// TwinCAT 3 PLC project Plc
// ProgramVersion: 3.1.4026.19
// libraries:
//   Tc2_Standard, * (Beckhoff Automation GmbH)
//   Tc2_System, * (Beckhoff Automation GmbH)
//   TcUnit, * (www.tcunit.org)
// project tree:
//   / CCTask1.TcTTO, CCTask2.TcTTO, PlcTask.TcTTO
//   Program/ MAIN.TcPOU
//   Src/Base/ FB_VarByteBufferBase.TcPOU, I_VarByteBufferBase.TcIO
//   Src/SimpleDynBuffer/ FB_SimpleRingBuffer.TcPOU, I_SimpleRingBuffer.TcIO
//   Src/ThreadSafe/ FB_SpscBuffer.TcPOU, I_SpscBuffer.TcIO
//   Src/VarByteBuffer/ FB_VarByteBuffer.TcPOU, I_VarByteBuffer.TcIO
//   Src/VarStringBuffer/ FB_VarStringBuffer.TcPOU, I_VarStringBuffer.TcIO
//   _test/SimpleRingBuffer/DUT/ ST_TestStruct.TcDUT
//   _test/SimpleRingBuffer/ FB_TestSimpleDynBuffer.TcPOU
//   _test/ThreadSafe/ ProgramTask1.TcPOU, ProgramTask2.TcPOU
//   _test/VarStringBuffer/ FB_TestVarStringBuffer.TcPOU
// real-time tasks:
//   TASK PlcTask: cycle T#30ms, priority 20, ADS port 350
//   TASK CCTask1: cycle T#2ms, priority 1, ADS port 351
//   TASK CCTask2: cycle T#3ms, priority 2, ADS port 352

CONFIGURATION Plc
    RESOURCE PLC ON TwinCAT3
        TASK CCTask1(INTERVAL := T#2ms, PRIORITY := 1);
        TASK CCTask2(INTERVAL := T#3ms, PRIORITY := 2);
        TASK PlcTask(INTERVAL := T#30ms, PRIORITY := 20);
        PROGRAM ProgramTask1 WITH CCTask1 : ProgramTask1;
        PROGRAM ProgramTask2 WITH CCTask2 : ProgramTask2;
        PROGRAM MAIN WITH PlcTask : MAIN;
    END_RESOURCE
END_CONFIGURATION

// ---- _test/SimpleRingBuffer/DUT/ST_TestStruct.TcDUT
TYPE ST_TestStruct :
STRUCT
	nIndex: UDINT;
	aData : ARRAY[1..1020] OF BYTE;
END_STRUCT
END_TYPE

// ---- Src/Base/I_VarByteBufferBase.TcIO
INTERFACE I_VarByteBufferBase

PROPERTY Buffer : PVOID
GET
END_GET
END_PROPERTY

PROPERTY Capacity : UDINT
GET
END_GET
END_PROPERTY

METHOD Clear : BOOL
END_METHOD

PROPERTY FreeBytes : UDINT
GET
END_GET
END_PROPERTY

METHOD Initialize : BOOL
VAR_INPUT
	nBufferSize 		: UDINT; // Size in byte
END_VAR
END_METHOD

METHOD Reset
END_METHOD

PROPERTY Size : UDINT
GET
END_GET
END_PROPERTY

END_INTERFACE

// ---- Src/SimpleDynBuffer/I_SimpleRingBuffer.TcIO
INTERFACE I_SimpleRingBuffer

PROPERTY Capacity : UDINT
GET
END_GET
END_PROPERTY

PROPERTY Empty : bool
GET
END_GET
END_PROPERTY

PROPERTY Full : bool
GET
END_GET
END_PROPERTY

METHOD Get : BOOL
VAR_INPUT
	pDestination 	: pvoid;
	cbSize 			: UDINT;
END_VAR
END_METHOD

METHOD Initialize : BOOL
VAR_INPUT
	nElementSize 		: UDINT;
	nElementCapacity 	: UDINT;
END_VAR
END_METHOD

METHOD Push : BOOL
VAR_INPUT
	pData : pvoid;
	cbSize : UDINT;
END_VAR
END_METHOD

METHOD Reset
END_METHOD

PROPERTY Size : UDINT
GET
END_GET
END_PROPERTY

END_INTERFACE

// ---- Src/ThreadSafe/I_SpscBuffer.TcIO
INTERFACE I_SpscBuffer

PROPERTY Capacity : UDINT
GET
END_GET
END_PROPERTY

METHOD Clear
VAR_INPUT
END_VAR
END_METHOD

PROPERTY Empty : bool
GET
END_GET
END_PROPERTY

PROPERTY Full : bool
GET
END_GET
END_PROPERTY

METHOD Get : BOOL
VAR_INPUT
	pDestination 	: pvoid;
	cbSize 			: UDINT;
END_VAR
END_METHOD

METHOD Initialize : BOOL
VAR_INPUT
	nElementSize 		: UDINT;
	nElementCapacity 	: UDINT;
END_VAR
END_METHOD

METHOD Push : BOOL
VAR_INPUT
	pData : pvoid;
	cbSize : UDINT;
END_VAR
END_METHOD

METHOD Reset
END_METHOD

PROPERTY Size : UDINT
GET
END_GET
END_PROPERTY

END_INTERFACE

// ---- Src/VarByteBuffer/I_VarByteBuffer.TcIO
INTERFACE I_VarByteBuffer EXTENDS I_VarByteBufferBase

METHOD Push : BOOL
VAR_INPUT
	pData : pvoid;
	cbSize : UDINT;
END_VAR
END_METHOD

END_INTERFACE

// ---- Src/VarStringBuffer/I_VarStringBuffer.TcIO
INTERFACE I_VarStringBuffer EXTENDS I_VarByteBufferBase

METHOD Push : BOOL
VAR_INPUT
	sInputString	: REFERENCE TO T_MaxString;
END_VAR
END_METHOD

END_INTERFACE

// ---- _test/ThreadSafe/ProgramTask1.TcPOU
PROGRAM ProgramTask1
VAR
	fbSpscBuff 	: FB_SpscBuffer;
	ipSpscBuff 	: I_SpscBuffer 		:= fbSpscBuff;
	nCounter 	: UDINT;
	bInit 		: BOOL;
END_VAR

nCounter := nCounter + 1;
IF NOT(binit) THEN
	bInit := TRUE;
	ipSpscBuff.Initialize(SIZEOF(UDINT),100);
END_IF

ipSpscBuff.Push(ADR(nCounter),SIZEOF(nCounter));
ipSpscBuff.Reset();

END_PROGRAM

// ---- Src/ThreadSafe/FB_SpscBuffer.TcPOU
FUNCTION_BLOCK FB_SpscBuffer IMPLEMENTS I_SpscBuffer
VAR
	_pBuffer 		: POINTER TO BYTE;
	_nTail 			: UDINT;
	_nHead 			: UDINT;
	_nCapacity 		: UDINT;
	_bFull 			: BOOL;
	_nSize 			: UDINT;
	
	_fbCriticalSection : FB_IecCriticalSection;
	_nElementSize 	: UDINT;
	_nLockFailures	: UDINT;
	_nError 		: UDINT;
END_VAR
VAR CONSTANT
	cMaxElementSize : UDINT := 4096;
END_VAR

PROPERTY Capacity : UDINT
GET
Capacity := this^._nCapacity;
END_GET
END_PROPERTY

METHOD Clear
VAR_INPUT
END_VAR
IF THIS^._fbCriticalSection.Enter() THEN
	THIS^._nTail 			:= 0;
	THIS^._nHead 			:= 0;
	THIS^._nCapacity 		:= 0;
	THIS^._bFull 			:= 0;
	THIS^._nSize 			:= 0;
	THIS^._nElementSize 	:= 0;
	THIS^._nError 			:= 0;
	THIS^._fbCriticalSection.Leave();
ELSE
	THIS^._nLockFailures := THIS^._nLockFailures :=  + 1;
	RETURN;
END_IF
END_METHOD

PROPERTY Empty : bool
GET
Empty := not(this^._bFull) and (this^._nHead = this^._nTail);
END_GET
END_PROPERTY

//FB_Exit must be implemented explicitly. If there is an implementation, then the
//method is called before the controller removes the code of the function block instance
//(implicit call). The return value is not evaluated.
METHOD FB_Exit: BOOL
VAR_INPUT
    bInCopyCode: BOOL;  // TRUE: the exit method is called in order to leave the instance which will be copied afterwards (online change).  
END_VAR
this^.Reset();
END_METHOD

PROPERTY Full : bool
GET
Full := this^._bFull;
END_GET
END_PROPERTY

METHOD Get : BOOL
VAR_INPUT
	pDestination 	: pvoid;
	cbSize 			: UDINT;
END_VAR
VAR
	nByteOffset : UDINT;
	res 		: UDINT;
END_VAR
IF THIS^._fbCriticalSection.Enter() THEN
	IF (THIS^._pBuffer = 0) OR (THIS^._nCapacity = 0) THEN  RETURN; END_IF; 	// Check initialization
	IF pDestination = 0 THEN  RETURN; END_IF;								// Check input
	IF cbSize <> THIS^._nElementSize THEN  RETURN; END_IF;					// Check input
	IF THIS^.Empty THEN RETURN; END_IF;										// Check internal state
	
	nByteOffset := THIS^._nTail*THIS^._nElementSize;
	res := memcpy(pDestination, THIS^._pBuffer + nByteOffset, THIS^._nElementSize);
	
	IF res <> THIS^._nElementSize THEN
		THIS^._nError := THIS^._nError + 1;
	END_IF
	
	THIS^._bFull := FALSE;
	IF THIS^._nSize > 0 THEN
		THIS^._nSize := THIS^._nSize - 1;	
	END_IF
	THIS^._nTail := (THIS^._nTail + 1) MOD THIS^._nCapacity;
	
	THIS^._fbCriticalSection.Leave();
	Get := TRUE;

ELSE
	THIS^._nLockFailures := THIS^._nLockFailures :=  + 1;
	RETURN;
END_IF
END_METHOD

METHOD Initialize : BOOL
VAR_INPUT
	nElementSize 		: UDINT;
	nElementCapacity 	: UDINT;
END_VAR
VAR
	nSize 				: UDINT;
END_VAR
IF nElementSize = 0 OR nElementCapacity = 0 THEN RETURN; END_IF;
IF nElementSize > THIS^.cMaxElementSize THEN RETURN; END_IF;
IF (nElementCapacity > (TO_UDINT(16#FFFFFFFF) / nElementSize)) THEN RETURN; END_IF;

THIS^.Reset();

nSize := nElementSize * nElementCapacity;
THIS^._pBuffer := __NEW(BYTE, nSize);

IF THIS^._pBuffer = 0 THEN RETURN; END_IF;
THIS^._nElementSize := nElementSize;
THIS^._nCapacity := nElementCapacity;
Initialize := TRUE;
END_METHOD

METHOD Push : BOOL
VAR_INPUT
	pData : pvoid;
	cbSize : UDINT;
END_VAR
VAR
	nByteOffset : UDINT;
	res			: UDINT;
END_VAR
IF THIS^._fbCriticalSection.Enter() THEN
	
	IF (THIS^._pBuffer = 0) OR (THIS^._nCapacity = 0) THEN RETURN; END_IF;		// Check initialization
	IF THIS^._bFull THEN RETURN; END_IF;
	IF cbSize <> THIS^._nElementSize THEN RETURN; END_IF;						// Check input
	IF pData = 0 THEN RETURN; END_IF											// Check input
	
	nByteOffset := THIS^._nHead*THIS^._nElementSize;
	res := memcpy(THIS^._pBuffer + nByteOffset,pData,THIS^._nElementSize);
	IF res <> THIS^._nElementSize THEN
		THIS^._nError := THIS^._nError + 1; 
	END_IF	

	THIS^._nSize := THIS^._nSize + 1;

	
	THIS^._nHead := (THIS^._nHead + 1) MOD THIS^._nCapacity;
	THIS^._bFull := THIS^._nHead = THIS^._nTail;
	
	Push := TRUE;
	THIS^._fbCriticalSection.Leave();
	

ELSE
	THIS^._nLockFailures := THIS^._nLockFailures :=  + 1;
	RETURN;
END_IF
END_METHOD

METHOD Reset
IF THIS^._fbCriticalSection.Enter() THEN
	IF THIS^._pBuffer <> 0 THEN
		__DELETE(THIS^._pBuffer);
		THIS^._pBuffer := 0;
	END_IF
	
	THIS^._nTail 			:= 0;
	THIS^._nHead 			:= 0;
	THIS^._nCapacity 		:= 0;
	THIS^._bFull 			:= 0;
	THIS^._nSize 			:= 0;
	THIS^._nElementSize 	:= 0;
	THIS^._nError 			:= 0;
	THIS^._fbCriticalSection.Leave();
ELSE
	THIS^._nLockFailures := THIS^._nLockFailures :=  + 1;
	RETURN;
END_IF
END_METHOD

PROPERTY Size : UDINT
GET
Size := (this^._nHead-this^._nTail + this^.Capacity) mod this^.Capacity;
END_GET
END_PROPERTY

END_FUNCTION_BLOCK

// ---- _test/ThreadSafe/ProgramTask2.TcPOU
PROGRAM ProgramTask2
VAR
	nRead : udint;
END_VAR

ProgramTask1.ipSpscBuff.Get(ADR(nRead),SIZEOF(nRead));

END_PROGRAM

// ---- Program/MAIN.TcPOU
PROGRAM MAIN
VAR
	nCounter 				: INT;
	fbTestSimpleDynBuffer 	: FB_TestSimpleDynBuffer;
	fbTestVarByteBuffer		: FB_TestVarStringBuffer;
END_VAR

nCounter := nCounter + 1;

TcUnit.RUN();

END_PROGRAM

// ---- _test/SimpleRingBuffer/FB_TestSimpleDynBuffer.TcPOU
FUNCTION_BLOCK FB_TestSimpleDynBuffer EXTENDS TcUnit.FB_TestSuite
VAR

	// FillTenElements
	fbBufferTest1 : FB_SimpleRingBuffer;
	ipBufferTest1 : I_SimpleRingBuffer := fbBufferTest1;

	//OverflowOneElement
	fbBufferTest2 : FB_SimpleRingBuffer;
	ipBufferTest2 : I_SimpleRingBuffer := fbBufferTest2;

	//ResetAndUse
	fbBufferTest3 : FB_SimpleRingBuffer;
	ipBufferTest3 : I_SimpleRingBuffer := fbBufferTest2;

	//CheckMemoryLeaks
	fbBufferTest4 	: FB_SimpleRingBuffer;
	ipBufferTest4 	: I_SimpleRingBuffer := fbBufferTest4;
	nState4 		: UDINT;
	nFillPerCycle 	: UDINT := 64;
	nKbToFill 		: UDINT := 10*1024;
	nFillCyclesToDo : UDINT := nKbToFill/nFillPerCycle; // 10 mb 
	nFillCycle 		: UDINT;
	nErrors4 		: UDINT;

	//CheckInvalidInput
	fbBufferTest5 : FB_SimpleRingBuffer;
	ipBufferTest5 : I_SimpleRingBuffer := fbBufferTest2;

END_VAR

FillTenElements();
OverflowOneElement();
ResetAndUse();
// CheckMemoryLeaks();
CheckInvalidInput();

METHOD CheckInvalidInput : REFERENCE TO FB_Test
VAR
	i 		: UDINT;
	nGet : UDINT;

END_VAR
TEST('CheckInvalidInput');


IF ipBufferTest5.Initialize(	nElementSize := 0,
								nElementCapacity := 1) THEN
	AssertTrue(FALSE, 'Failed init 0 element size');		
END_IF;

IF ipBufferTest5.Initialize(	nElementSize := 4,
								nElementCapacity := 0) THEN
	AssertTrue(FALSE, 'Failed init 0 capacity');		
END_IF;

IF NOT ipBufferTest5.Initialize(	nElementSize := 4,
									nElementCapacity := 1) THEN
	AssertTrue(FALSE, 'Failed init');		
END_IF;

IF ipBufferTest5.Push(ADR(i),0) THEN
	AssertTrue(FALSE, 'Failed push size 0');		
END_IF

IF ipBufferTest5.Push(0,4) THEN
	AssertTrue(FALSE, 'Failed push adr 0');		
END_IF

IF NOT ipBufferTest5.Push(ADR(i),4) THEN
	AssertTrue(FALSE, 'Failed push legit data');		
END_IF

IF ipBufferTest5.Get(ADR(i),0) THEN
	AssertTrue(FALSE, 'Failed get size 0');		
END_IF

IF ipBufferTest5.Get(0,4) THEN
	AssertTrue(FALSE, 'Failed get adr 0');		
END_IF

TEST_FINISHED();
END_METHOD

METHOD CheckMemoryLeaks : REFERENCE TO FB_Test
VAR
	i,j 				: UDINT;
	nElementsSize 		: UDINT;
	nOverflow			: UDINT 	:= 2;
	stDataToInsert		: ST_TestStruct; // 1024 bytes
	nElementsToPush		:UDINT;
	nReadSize 			: UDINT;
	bIsFull 			: BOOL;
	bIsEmpty 			: BOOL;
	nReadCapacity		: UDINT;
	
	nGetValue : ST_TestStruct;
	
	nExpectedValue : UDINT;
END_VAR
TEST('CheckMemoryLeaks');

CASE nState4 OF 
	0:

		nElementsSize := SIZEOF(ST_TestStruct);
		IF NOT fbBufferTest4.Initialize(	nElementSize := nElementsSize,
											nElementCapacity := 1024*10) THEN
 			nErrors4 := nErrors4 +1;
		END_IF;
		nState4 := 1;			
		

	1:
		IF nFillCycle = nFillCyclesToDo THEN
			nElementsToPush := nFillPerCycle + nOverflow;
		ELSE
			nElementsToPush := nFillPerCycle;
		END_IF
		FOR i := 1 TO nElementsToPush DO
			stDataToInsert.nIndex := i;
			IF NOT fbBufferTest4.Push(ADR(stDataToInsert), SIZEOF(stDataToInsert)) THEN
				nErrors4 := nErrors4 +1;
			END_IF
		END_FOR
		nFillCycle := nFillCycle + 1;
		IF nFillCycle >= nFillCyclesToDo THEN
			nFillCycle := 1;
			nState4 := 10;
		END_IF
	10:
		// Free cylce
		FOR i := 1 TO nFillPerCycle DO
			IF NOT fbBufferTest4.Get(ADR(nGetValue), SIZEOF(nGetValue)) THEN
				nErrors4 := nErrors4 +1;
			END_IF
		END_FOR

		nFillCycle := nFillCycle + 1;
		IF nFillCycle >= nFillCyclesToDo THEN
			fbBufferTest4.Reset();
			nFillCycle := 0;
			nState4 := 20;
		END_IF
	20: 
		
		bIsFull 	:= fbBufferTest4.Full;
		nReadSize 	:= fbBufferTest4.Size;
		nExpectedValue := 0;
		AssertFalse(bIsFull, 'Inconsistent Full flag');		
		AssertEquals(Expected 	:= nExpectedValue,
					 Actual 	:= nReadSize,
					 Message 	:= 'Error computing Size');		
		AssertEquals(Expected 	:= nExpectedValue,
					 Actual 	:= nErrors4,
					 Message 	:= 'Error computing Size');		
		TEST_FINISHED(); 
END_CASE
END_METHOD

METHOD FillTenElements : BOOL
VAR
	i 					: UDINT;
	nCapacity 			: UDINT 	:= 10;
	nElementsSize 		: UDINT;
	
	nReadSize 			: UDINT;
	bIsFull 			: BOOL;
	bIsEmpty 			: BOOL;
	nReadCapacity		: UDINT;
END_VAR
TEST('PushTenElements');

nElementsSize := SIZEOF(UDINT);
IF NOT ipBufferTest1.Initialize(	nElementSize := nElementsSize,
									nElementCapacity := nCapacity) THEN
	AssertTrue(FALSE, 'PushTenElements failed to initialize.');		
END_IF;

bIsEmpty := ipBufferTest1.Empty;
nReadCapacity := ipBufferTest1.Capacity;
AssertTrue(bIsEmpty, 'PushTenElements failed to initialize.');
AssertEquals(Expected 	:= nCapacity,
             Actual 	:= nReadCapacity,
             Message 	:= 'Error computing capacity');				
			 
FOR i := 1 TO nCapacity DO
	IF NOT ipBufferTest1.Push(ADR(i), SIZEOF(i)) THEN
		AssertTrue(FALSE, 'Failed to push');
	END_IF
END_FOR

bIsFull 	:= ipBufferTest1.Full;
nReadSize 	:= ipBufferTest1.Size;

AssertTrue(bIsFull, 'Inconsistent Full flag');		
AssertEquals(Expected 	:= nCapacity,
             Actual 	:= nReadSize,
             Message 	:= 'Error computing Size');		
 
TEST_FINISHED();
END_METHOD

METHOD OverflowOneElement : REFERENCE TO FB_Test
VAR
	i 					: UDINT;
	nCapacity 			: UDINT 	:= 10;
	nElementsSize 		: UDINT;
	nOverflow			: UDINT 	:= 1;
	
	nReadSize 			: UDINT;
	bIsFull 			: BOOL;
	bIsEmpty 			: BOOL;
	nReadCapacity		: UDINT;
	
	nGetValue : UDINT;
	
	nExpectedValue : UDINT;
END_VAR
TEST('OverflowOneElement');

nElementsSize := SIZEOF(UDINT);
IF NOT ipBufferTest2.Initialize(	nElementSize := nElementsSize,
									nElementCapacity := nCapacity) THEN
	AssertTrue(FALSE, 'PushTenElements failed to initialize.');		
END_IF;

bIsEmpty := ipBufferTest2.Empty;
nReadCapacity := ipBufferTest2.Capacity;
AssertTrue(bIsEmpty, 'PushTenElements failed to initialize.');
AssertEquals(Expected 	:= nCapacity,
             Actual 	:= nReadCapacity,
             Message 	:= 'Error computing capacity');				
			 
FOR i := 1 TO nCapacity + nOverflow DO
	IF NOT ipBufferTest2.Push(ADR(i), SIZEOF(i)) THEN
		AssertTrue(FALSE, 'Failed to push');
	END_IF
END_FOR
FOR i := 1 TO nCapacity DO
	IF NOT ipBufferTest2.Get(ADR(nGetValue), SIZEOF(nGetValue)) THEN
		AssertTrue(FALSE, 'Failed to get');
	ELSE
		nExpectedValue := i + nOverflow;
		AssertEquals(Expected 	:= nExpectedValue,
					 Actual 	:= nGetValue,
					 Message 	:= 'Error on Get');
	END_IF
END_FOR

bIsFull 	:= ipBufferTest2.Full;
nReadSize 	:= ipBufferTest2.Size;

nExpectedValue := 0;
AssertFalse(bIsFull, 'Inconsistent Full flag');		
AssertEquals(Expected 	:= nExpectedValue,
             Actual 	:= nReadSize,
             Message 	:= 'Error computing Size');		
 
TEST_FINISHED();
END_METHOD

METHOD ResetAndUse : REFERENCE TO FB_Test
VAR
	i,j 				: UDINT;
	nCapacity 			: UDINT 	:= 10;
	nElementsSize 		: UDINT;
	nOverflow			: UDINT 	:= 1;
	
	nReadSize 			: UDINT;
	bIsFull 			: BOOL;
	bIsEmpty 			: BOOL;
	nReadCapacity		: UDINT;
	
	nGetValue : UDINT;
	
	nExpectedValue : UDINT;
END_VAR
TEST('ResetAndUse');

FOR j := 1 TO 100 DO

	nElementsSize := SIZEOF(UDINT);
	IF NOT ipBufferTest3.Initialize(	nElementSize := nElementsSize,
										nElementCapacity := nCapacity) THEN
		AssertTrue(FALSE, 'Failed to initialize.');		
	END_IF;
	
	bIsEmpty := ipBufferTest3.Empty;
	nReadCapacity := ipBufferTest3.Capacity;
	AssertTrue(bIsEmpty, 'Failed to initialize.');
	AssertEquals(Expected 	:= nCapacity,
				 Actual 	:= nReadCapacity,
				 Message 	:= 'Error computing capacity');				
				 
	FOR i := 1 TO nCapacity + nOverflow DO
		IF NOT ipBufferTest3.Push(ADR(i), SIZEOF(i)) THEN
			AssertTrue(FALSE, 'Failed to push');
		END_IF
	END_FOR
	FOR i := 1 TO nCapacity DO
		IF NOT ipBufferTest3.Get(ADR(nGetValue), SIZEOF(nGetValue)) THEN
			AssertTrue(FALSE, 'Failed to get');
		ELSE
			nExpectedValue := i + nOverflow;
			AssertEquals(Expected 	:= nExpectedValue,
						 Actual 	:= nGetValue,
						 Message 	:= 'Error on Get');
		END_IF
	END_FOR
	
	bIsFull 	:= ipBufferTest3.Full;
	nReadSize 	:= ipBufferTest3.Size;
	
	nExpectedValue := 0;
	AssertFalse(bIsFull, 'Inconsistent Full flag');		
	AssertEquals(Expected 	:= nExpectedValue,
				 Actual 	:= nReadSize,
				 Message 	:= 'Error computing Size');		
	ipBufferTest3.Reset();
END_FOR
TEST_FINISHED();
END_METHOD

END_FUNCTION_BLOCK

// ---- Src/SimpleDynBuffer/FB_SimpleRingBuffer.TcPOU
FUNCTION_BLOCK FB_SimpleRingBuffer implements I_SimpleRingBuffer
VAR
	_pBuffer 		: POINTER TO BYTE;
	_nTail 			: UDINT;
	_nHead 			: UDINT;
	_nCapacity 		: UDINT;
	_bFull 			: BOOL;
	_nSize 			: UDINT;
	
	_nElementSize 	: UDINT;
	_nError 		: UDINT;
END_VAR
VAR CONSTANT
	cMaxElementSize : UDINT := 4096;
END_VAR

PROPERTY Capacity : UDINT
GET
Capacity := this^._nCapacity;
END_GET
END_PROPERTY

PROPERTY Empty : bool
GET
Empty := not(this^._bFull) and (this^._nHead = this^._nTail);
END_GET
END_PROPERTY

//FB_Exit must be implemented explicitly. If there is an implementation, then the
//method is called before the controller removes the code of the function block instance
//(implicit call). The return value is not evaluated.
METHOD FB_Exit: BOOL
VAR_INPUT
    bInCopyCode: BOOL;  // TRUE: the exit method is called in order to leave the instance which will be copied afterwards (online change).  
END_VAR
this^.Reset();
END_METHOD

PROPERTY Full : bool
GET
Full := this^._bFull;
END_GET
END_PROPERTY

METHOD Get : BOOL
VAR_INPUT
	pDestination 	: pvoid;
	cbSize 			: UDINT;
END_VAR
VAR
	nByteOffset : UDINT;
	res 		: UDINT;
END_VAR
IF (THIS^._pBuffer = 0) OR (THIS^._nCapacity = 0) THEN RETURN; END_IF; 	// Check initialization
IF pDestination = 0 THEN RETURN; END_IF;								// Check input
IF cbSize <> THIS^._nElementSize THEN RETURN; END_IF;					// Check input
IF THIS^.Empty THEN RETURN; END_IF;										// Check internal state

nByteOffset := THIS^._nTail*THIS^._nElementSize;
res := memcpy(pDestination, THIS^._pBuffer + nByteOffset, THIS^._nElementSize);

IF res <> THIS^._nElementSize THEN
	THIS^._nError := THIS^._nError + 1;
	RETURN;
END_IF

THIS^._bFull := FALSE;
IF THIS^._nSize > 0 THEN
	THIS^._nSize := THIS^._nSize - 1;	
END_IF
THIS^._nTail := (THIS^._nTail + 1) MOD THIS^._nCapacity;

Get := TRUE;
END_METHOD

METHOD Initialize : BOOL
VAR_INPUT
	nElementSize 		: UDINT;
	nElementCapacity 	: UDINT;
END_VAR
VAR
	nSize 				: UDINT;
END_VAR
IF nElementSize = 0 OR nElementCapacity = 0 THEN RETURN; END_IF;
IF nElementSize > THIS^.cMaxElementSize THEN RETURN; END_IF;
IF (nElementCapacity > (TO_UDINT(16#FFFFFFFF) / nElementSize)) THEN RETURN; END_IF;

THIS^.Reset();

nSize := nElementSize * nElementCapacity;
THIS^._pBuffer := __NEW(BYTE, nSize);

IF THIS^._pBuffer = 0 THEN RETURN; END_IF;
THIS^._nElementSize := nElementSize;
THIS^._nCapacity := nElementCapacity;
Initialize := TRUE;
END_METHOD

METHOD Push : BOOL
VAR_INPUT
	pData : pvoid;
	cbSize : UDINT;
END_VAR
VAR
	nByteOffset : UDINT;
	res			: UDINT;
END_VAR
IF (THIS^._pBuffer = 0) OR (THIS^._nCapacity = 0) THEN RETURN; END_IF;		// Check initialization
IF cbSize <> THIS^._nElementSize THEN RETURN; END_IF;						// Check input
IF pData = 0 THEN RETURN; END_IF											// Check input

nByteOffset := THIS^._nHead*THIS^._nElementSize;
res := memcpy(THIS^._pBuffer + nByteOffset,pData,THIS^._nElementSize);
IF res <> THIS^._nElementSize THEN
	THIS^._nError := THIS^._nError + 1; 
	RETURN;
END_IF

IF THIS^._bFull THEN
	THIS^._nTail := (THIS^._nTail + 1) MOD THIS^._nCapacity;
ELSE
	THIS^._nSize := THIS^._nSize + 1;
END_IF

THIS^._nHead := (THIS^._nHead + 1) MOD THIS^._nCapacity;
THIS^._bFull := THIS^._nHead = THIS^._nTail;

Push := TRUE;
END_METHOD

METHOD Reset
IF THIS^._pBuffer <> 0 THEN
	__DELETE(THIS^._pBuffer);
	THIS^._pBuffer := 0;
END_IF

THIS^._nTail 			:= 0;
THIS^._nHead 			:= 0;
THIS^._nCapacity 		:= 0;
THIS^._bFull 			:= 0;
THIS^._nSize 			:= 0;
THIS^._nElementSize 	:= 0;
THIS^._nError 			:= 0;
END_METHOD

PROPERTY Size : UDINT
GET
Size := this^._nSize;
END_GET
END_PROPERTY

END_FUNCTION_BLOCK

// ---- _test/VarStringBuffer/FB_TestVarStringBuffer.TcPOU
FUNCTION_BLOCK FB_TestVarStringBuffer EXTENDS TcUnit.FB_TestSuite
VAR
	fbTestBuffer1 : FB_VarStringBuffer;
	ipTestBuffer1 : I_VarStringBuffer	:= fbTestBuffer1;
	
	fbTestBuffer2 : FB_VarStringBuffer;
	ipTestBuffer2 : I_VarStringBuffer	:= fbTestBuffer2;
	
	fbTestBuffer3 : FB_VarStringBuffer;
	ipTestBuffer3 : I_VarStringBuffer	:= fbTestBuffer3;
END_VAR

CommonUseCase();
ValidateInput();
BlockWhenFull();

METHOD BlockWhenFull : REFERENCE TO FB_Test
VAR
	cBufferSize 		: UDINT := 22;
	cNumberOfElements 	: UDINT := 5;
	cOutBufferSize 		: UDINT := 22;
	cExpectedFreeBytes 	: UDINT := 2;
	
	aInElements : ARRAY[1..6] OF T_MaxString := [	'AAAAA','BBBBB','CCCCC','DDDDD','EEEEE'];
	
	sOutBuffer 	: STRING(22);
	i 			: UDINT;
	res 		: UDINT;
	
	nReadCapacity 	: UDINT;
	nReadBuffer 	: PVOID;
	nReadFreeBytes 	: UDINT;
	bIsNotZero 		: BOOL;
END_VAR
TEST('BlockWhenFull');
ipTestBuffer3.Initialize(cBufferSize);

FOR i := 1 TO cNumberOfElements DO
	ipTestBuffer3.Push(aInElements[i]);
END_FOR

IF ipTestBuffer3.Push(aInElements[5]) THEN
	AssertTrue(FALSE, 'Memory Corrupted');	
END_IF

nReadCapacity 	:= ipTestBuffer3.Capacity;
nReadFreeBytes 	:= ipTestBuffer3.FreeBytes;

AssertEquals(Expected 	:= cBufferSize,
             Actual 	:= nReadCapacity,
             Message 	:= 'Error computing Capacity');
	
			 
AssertEquals(Expected 	:= cExpectedFreeBytes,
             Actual 	:= nReadFreeBytes,
             Message 	:= 'Error computing FreeBytes'); 
			 
						
res := memcpy(ADR(sOutBuffer), ipTestBuffer3.Buffer, SIZEOF(sOutBuffer));

AssertEquals_STRING(	Expected := 'AAAAABBBBBCCCCCDDDDD',
						Actual := sOutBuffer,
						Message := 'Error extracting the buffer');
			 
						
TEST_FINISHED();
END_METHOD

METHOD CommonUseCase : REFERENCE TO FB_Test
VAR
	cBufferSize 		: UDINT := 20;
	cNumberOfElements 	: UDINT := 5;
	cOutBufferSize 		: UDINT := 17;
	cExpectedFreeBytes 	: UDINT := 3;
	
	aInElements : ARRAY[1..5] OF T_MaxString := [	'AAAAAA','BBBBB','CCC','DD','E'];
	
	sOutBuffer 	: STRING(20);
	i 			: UDINT;
	res 		: UDINT;
	
	nReadCapacity 	: UDINT;
	nReadBuffer 	: PVOID;
	nReadFreeBytes 	: UDINT;
	bIsNotZero 		: BOOL;
END_VAR
TEST('CommonUseCase');
IF NOT ipTestBuffer1.Initialize(cBufferSize) THEN
	AssertTrue(FALSE, 'Failed to initialize.');		
END_IF

FOR i := 1 TO cNumberOfElements DO
	ipTestBuffer1.Push(aInElements[i]);
END_FOR

nReadCapacity 	:= ipTestBuffer1.Capacity;
nReadBuffer 	:= ipTestBuffer1.Buffer;
nReadFreeBytes 	:= ipTestBuffer1.FreeBytes;
bIsNotZero := nReadBuffer <> 0;

AssertEquals(Expected 	:= cBufferSize,
             Actual 	:= nReadCapacity,
             Message 	:= 'Error computing Capacity');

AssertTrue(bIsNotZero, 'Failed to allocate the buffer');		
			 
AssertEquals(Expected 	:= cExpectedFreeBytes,
             Actual 	:= nReadFreeBytes,
             Message 	:= 'Error computing FreeBytes'); 
			 
						
res := memcpy(ADR(sOutBuffer), nReadBuffer, SIZEOF(sOutBuffer));

AssertEquals_STRING(	Expected := 'AAAAAABBBBBCCCDDE',
						Actual := sOutBuffer,
						Message := 'Error extracting the buffer');
						
IF NOT ipTestBuffer1.Clear() THEN
	AssertTrue(FALSE, 'Failed to clear');		
END_IF

nReadCapacity 	:= ipTestBuffer1.Capacity;
nReadBuffer 	:= ipTestBuffer1.Buffer;
nReadFreeBytes 	:= ipTestBuffer1.FreeBytes;
bIsNotZero := nReadBuffer <> 0;

AssertEquals(Expected 	:= cBufferSize,
             Actual 	:= nReadCapacity,
             Message 	:= 'Error computing Capacity after clear');

AssertTrue(bIsNotZero, 'Buffer Corrupted after clear');		
			 
AssertEquals(Expected 	:= cBufferSize,
             Actual 	:= nReadFreeBytes,
             Message 	:= 'Error computing FreeBytes after clear'); 
			 
						
TEST_FINISHED();
END_METHOD

METHOD ValidateInput : REFERENCE TO FB_Test
VAR
	cBufferSize		: UDINT := 20;
	sString 		: T_MaxString := 'foo';
	sInvalidString 	: REFERENCE TO T_MaxString;
END_VAR
TEST('ValidateInput');

IF ipTestBuffer2.Push(sString) THEN
	AssertTrue(FALSE, 'Memory corrupted.');		
END_IF

ipTestBuffer2.Initialize(cBufferSize);

IF ipTestBuffer2.Push(sInvalidString) THEN
	AssertTrue(FALSE, 'Memory corrupted from invalid reference.');		
END_IF

TEST_FINISHED();
END_METHOD

END_FUNCTION_BLOCK

// ---- Src/VarStringBuffer/FB_VarStringBuffer.TcPOU
FUNCTION_BLOCK FB_VarStringBuffer EXTENDS FB_VarByteBufferBase IMPLEMENTS I_VarStringBuffer

METHOD Push : BOOL
VAR_INPUT
	sInputString	: REFERENCE TO T_MaxString;
END_VAR
VAR
	res 		: UDINT;
	nStringSize : UDINT;
END_VAR
IF (THIS^._pBuffer = 0) OR (THIS^._nCapacity = 0) THEN RETURN; END_IF;		// Check initialization
IF NOT __ISVALIDREF(sInputString) THEN RETURN; END_IF;

nStringSize := INT_TO_UDINT(len(sInputString));
IF nStringSize > THIS^.FreeBytes THEN RETURN; END_IF;

res := memcpy(THIS^._pBuffer + THIS^._nHead,ADR(sInputString),nStringSize);
IF res <> nStringSize THEN
	THIS^._nError := THIS^._nError + 1; 
	RETURN;
END_IF

THIS^._nHead := THIS^._nHead + nStringSize;
Push := TRUE;
END_METHOD

END_FUNCTION_BLOCK

// ---- Src/Base/FB_VarByteBufferBase.TcPOU
FUNCTION_BLOCK FB_VarByteBufferBase IMPLEMENTS I_VarByteBufferBase
VAR
	_pBuffer 		: POINTER TO BYTE;
	_nHead 			: UDINT;
	_nCapacity 		: UDINT;
	
	_nError			: UDINT;
END_VAR
VAR CONSTANT
	cMaxBufferSize 	: UDINT := 104857600 ; // 100 Mb
END_VAR

PROPERTY Buffer : PVOID
GET
Buffer := THIS^._pBuffer;
END_GET
END_PROPERTY

PROPERTY Capacity : UDINT
GET
Capacity := this^._nCapacity;
END_GET
END_PROPERTY

METHOD Clear : BOOL
VAR
	res : UDINT;
END_VAR
res := MEMSET(THIS^.Buffer, 0, THIS^.Capacity);
IF res <> THIS^.Capacity THEN RETURN; END_IF;
THIS^._nHead := 0;
Clear := TRUE;
END_METHOD

//FB_Exit must be implemented explicitly. If there is an implementation, then the
//method is called before the controller removes the code of the function block instance
//(implicit call). The return value is not evaluated.
METHOD FB_Exit: BOOL
VAR_INPUT
    bInCopyCode: BOOL;  // TRUE: the exit method is called in order to leave the instance which will be copied afterwards (online change).  
END_VAR
this^.Reset();
END_METHOD

PROPERTY FreeBytes : UDINT
GET
FreeBytes := THIS^._nCapacity - this^._nHead;
END_GET
END_PROPERTY

METHOD Initialize : BOOL
VAR_INPUT
	nBufferSize 		: UDINT; // Size in byte
END_VAR
IF nBufferSize = 0 OR nBufferSize > THIS^.cMaxBufferSize THEN RETURN; END_IF;

THIS^.Reset();

THIS^._nCapacity := nBufferSize;
THIS^._pBuffer := __NEW(BYTE, nBufferSize);
IF THIS^._pBuffer = 0 THEN RETURN; END_IF;

Initialize := TRUE;
END_METHOD

METHOD Reset
IF THIS^._pBuffer <> 0 THEN
	__DELETE(THIS^._pBuffer);
	THIS^._pBuffer := 0;
END_IF

THIS^._nHead 			:= 0;
THIS^._nCapacity 		:= 0;
THIS^._nError 			:= 0;
END_METHOD

PROPERTY Size : UDINT
GET
Size := this^._nHead;
END_GET
END_PROPERTY

END_FUNCTION_BLOCK

// ---- Src/VarByteBuffer/FB_VarByteBuffer.TcPOU
FUNCTION_BLOCK FB_VarByteBuffer EXTENDS FB_VarByteBufferBase IMPLEMENTS I_VarByteBuffer
VAR
END_VAR

METHOD Push : BOOL
VAR_INPUT
	pData : pvoid;
	cbSize : UDINT;
END_VAR
VAR;
	res			: UDINT;
END_VAR
IF (THIS^._pBuffer = 0) OR (THIS^._nCapacity = 0) THEN RETURN; END_IF;		// Check initialization
IF pData = 0 THEN RETURN; END_IF											// Check input
IF THIS^.FreeBytes < cbSize THEN RETURN; END_IF;

res := memcpy(THIS^._pBuffer + THIS^._nHead,pData,cbSize);
IF res <> cbSize THEN
	THIS^._nError := THIS^._nError + 1; 
	RETURN;
END_IF

THIS^._nHead := THIS^._nHead + cbSize;

Push := TRUE;
END_METHOD

END_FUNCTION_BLOCK
